SUBAPPLICATION logiBUS_PI_Speed_Publish_OPC (* logiBUS_PI_IDA (Puls-Eingang) als Frequenz (Hz) UND als bereits umgerechneter physikalischer Wert (km/h bzw. U/min, feste Skalierung) per OPC-UA publizieren, OHNE jegliche VT-Interaktion. Erweiterung von logiBUS_PI_Raw_Publish_OPC um die Hz->Einheit-Umrechnung (bisher zentral auf STG1 via AR_HZ_TO_Q_Publish_OPC) - jetzt lokal auf der Sensor-Station: der Rohwert (Hz) geht weiterhin nur ans Dashboard/Diagnose, verteilt wird nur noch der fertige physikalische Endwert. *)
  (* Standard: 61499-2; Description: Copyright (c) 2026 Meisterschulen am Ostbahnhof This program and the accompanying materials are made available under the terms of the Eclipse Public License 2.0 which is available at https://www.eclipse.org/legal/epl-2.0/ SPDX-License-Identifier: EPL-2.0 *)
  (* Version 1.0, 2026-09-17, Franz Höpfinger, Meisterschulen am Ostbahnhof, initial implementation - Franz: 'die Impulseingaenge will ich auch die Umrechnung auf dem Quellgeraet haben'. Erweitert logiBUS_PI_Raw_Publish_OPC (Rohwert-Kette: logiBUS_PI_IDA -> AD_TO_AR_NUM -> FT_DERIV_10_AR -> FT_PT1_AR, unveraendert) um AR_SPLIT_2 + initval_AR(SCALE) + AR_MUL_2 + zweite AR_PUBLISH_1-Instanz fuer den umgerechneten physikalischen Endwert - analog zum bisherigen AR_HZ_TO_Q_Publish_OPC-Muster (STG1), jetzt aber co-located mit dem Sensor statt zentral. *)
  PACKAGE MyLib::sys;
  IMPORT logiBUS::io::PI::logiBUS_PI;
  IMPORT logiBUS::io::PI::logiBUS_PI_S;
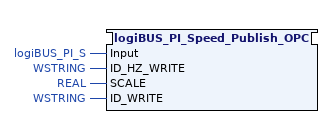
  VAR_INPUT
    Input : logiBUS::io::PI::logiBUS_PI_S := logiBUS_PI::Invalid; (* Identify the Input PulseInput_I1..I9 *)
    ID_HZ_WRITE : WSTRING; (* Frequenz-Publish-Adresse (REAL Hz, ACTION=PUBLISH) - nur fuer Dashboard/Diagnose, kein anderes Modul soll dies remote-abonnieren *)
    SCALE : REAL; (* Skalierungsfaktor Hz -> physikalische Einheit (z.B. 3.6/53 fuer km/h, 60.0 fuer U/min bei 1 Impuls/Umdrehung) *)
    ID_WRITE : WSTRING; (* Publish-Adresse des umgerechneten physikalischen Endwerts (REAL, ACTION=PUBLISH) - das ist die Adresse, die andere Stationen remote abonnieren *)
  END_VAR
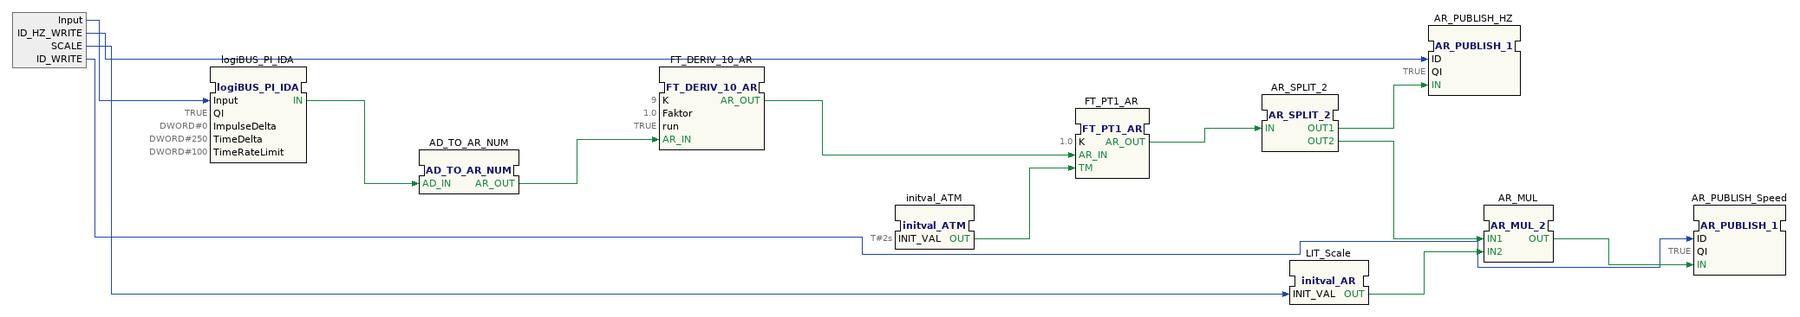
  FBS
    logiBUS_PI_IDA : logiBUS::io::PI::logiBUS_PI_IDA(QI := TRUE, ImpulseDelta := DWORD#0, TimeDelta := DWORD#250, TimeRateLimit := DWORD#100);
    AD_TO_AR_NUM : adapter::conversion::unidirectional::AD_TO_AR_NUM;
    FT_DERIV_10_AR : OSCAT_adapter::Control::FT_DERIV_10_AR(K := 9, Faktor := 1.0, run := TRUE);
    FT_PT1_AR : OSCAT_adapter::Control::FT_PT1_AR(K := 1.0);
    initval_ATM : adapter::types::unidirectional::ATM::initval::initval_ATM(INIT_VAL := T#2s);
    AR_SPLIT_2 : adapter::events::unidirectional::AR_SPLIT_2;
    AR_PUBLISH_HZ : adapter::net::AR_PUBLISH_1(QI := TRUE);
    LIT_Scale : adapter::types::unidirectional::AR::initval::initval_AR;
    AR_MUL : adapter::iec61131::arithmetic::AR_MUL_2;
    AR_PUBLISH_Speed : adapter::net::AR_PUBLISH_1(QI := TRUE);
  END_FBS
  DATA_CONNECTIONS
    Input TO logiBUS_PI_IDA.Input;
    ID_HZ_WRITE TO AR_PUBLISH_HZ.ID;
    SCALE TO LIT_Scale.INIT_VAL;
    ID_WRITE TO AR_PUBLISH_Speed.ID;
  END_CONNECTIONS
  ADAPTER_CONNECTIONS
    logiBUS_PI_IDA.IN TO AD_TO_AR_NUM.AD_IN;
    AD_TO_AR_NUM.AR_OUT TO FT_DERIV_10_AR.AR_IN;
    FT_DERIV_10_AR.AR_OUT TO FT_PT1_AR.AR_IN;
    initval_ATM.OUT TO FT_PT1_AR.TM;
    FT_PT1_AR.AR_OUT TO AR_SPLIT_2.IN;
    AR_SPLIT_2.OUT1 TO AR_PUBLISH_HZ.IN;
    AR_SPLIT_2.OUT2 TO AR_MUL.IN1;
    LIT_Scale.OUT TO AR_MUL.IN2;
    AR_MUL.OUT TO AR_PUBLISH_Speed.IN;
  END_CONNECTIONS
END_SUBAPPLICATION
